// TIA Portal V20 export
TYPE "SEW_MOVIKIT_VelocityDrive_STATUS_V2.1"
   STRUCT
      x_Bit_8_Fault : Bool;
      x_Bit_9_Warning : Bool;
      x_Bit_10_DriveTrain2_active : Bool;
      x_Bit_11_Setp_actual_speed_comp_signal_active : Bool;
      x_Bit_12_SW_Limit_switches_inactive : Bool;
      x_Bit_13_Reserved : Bool;
      x_Bit_14_StandBy_Mode_active : Bool;
      x_Bit_15_Heartbeat_OUT : Bool;
      x_Bit_0_Ready : Bool;
      x_Bit_1_STO_inactive : Bool;
      x_Bit_2_Output_Stage_enabled : Bool;
      x_Bit_3_Brake_released : Bool;
      x_Bit_4_Motor_turning : Bool;
      x_Bit_5_Active_Drive_referenced : Bool;
      x_Bit_6_New_Relative_Position_applied : Bool;
      x_Bit_7_In_Position : Bool;
      iActual_Speed : Int;
      wStatus_main_fault_sub_fault { ExternalAccessible := 'False'; ExternalVisible := 'False'; ExternalWritable := 'False'} : Word;
      iActual_Torque : Int;
      wDigital_Inputs : Word;
      bStatus_Fault : Byte;
      bStatus_subFault : Byte;
   END_STRUCT;
END_TYPE
